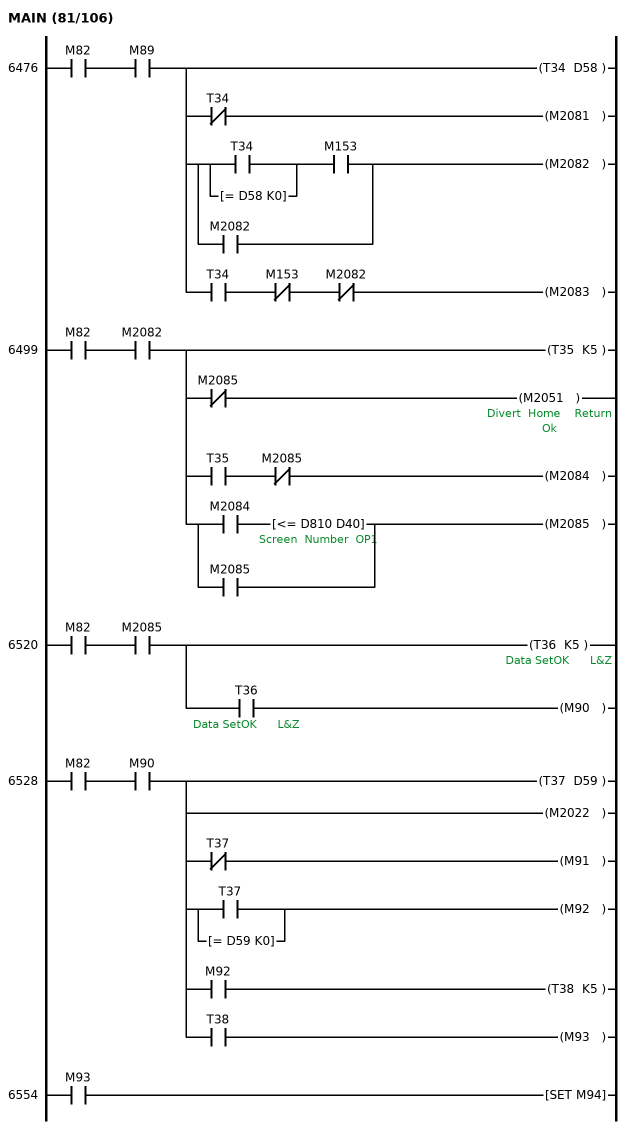
[picture p360: ladder of MAIN, rungs at steps 6476 to 6554]
6476  LD      M82
      AND     M89
      OUT     T34 D58
      MPS
      ANI     T34
      OUT     M2081
      MRD
      LD      T34
      OR=     D58 K0
      AND     M153
      OR      M2082
      ANB
      OUT     M2082
      MPP
      AND     T34
      ANI     M153
      ANI     M2082
      OUT     M2083
6499  LD      M82
      AND     M2082
      OUT     T35 K5
      MPS
      ANI     M2085
      OUT     M2051  ; Divert  Home    Return  Ok
      MRD
      AND     T35
      ANI     M2085
      OUT     M2084
      MPP
      LD      M2084
      AND<=   D810 D40  ; Screen  Number  OP1
      OR      M2085
      ANB
      OUT     M2085
6520  LD      M82
      AND     M2085
      OUT     T36 K5  ; Data SetOK      L&Z
      AND     T36  ; Data SetOK      L&Z
      OUT     M90
6528  LD      M82
      AND     M90
      OUT     T37 D59
      OUT     M2022
      MPS
      ANI     T37
      OUT     M91
      MRD
      LD      T37
      OR=     D59 K0
      ANB
      OUT     M92
      MRD
      AND     M92
      OUT     T38 K5
      MPP
      AND     T38
      OUT     M93
6554  LD      M93
      SET     M94
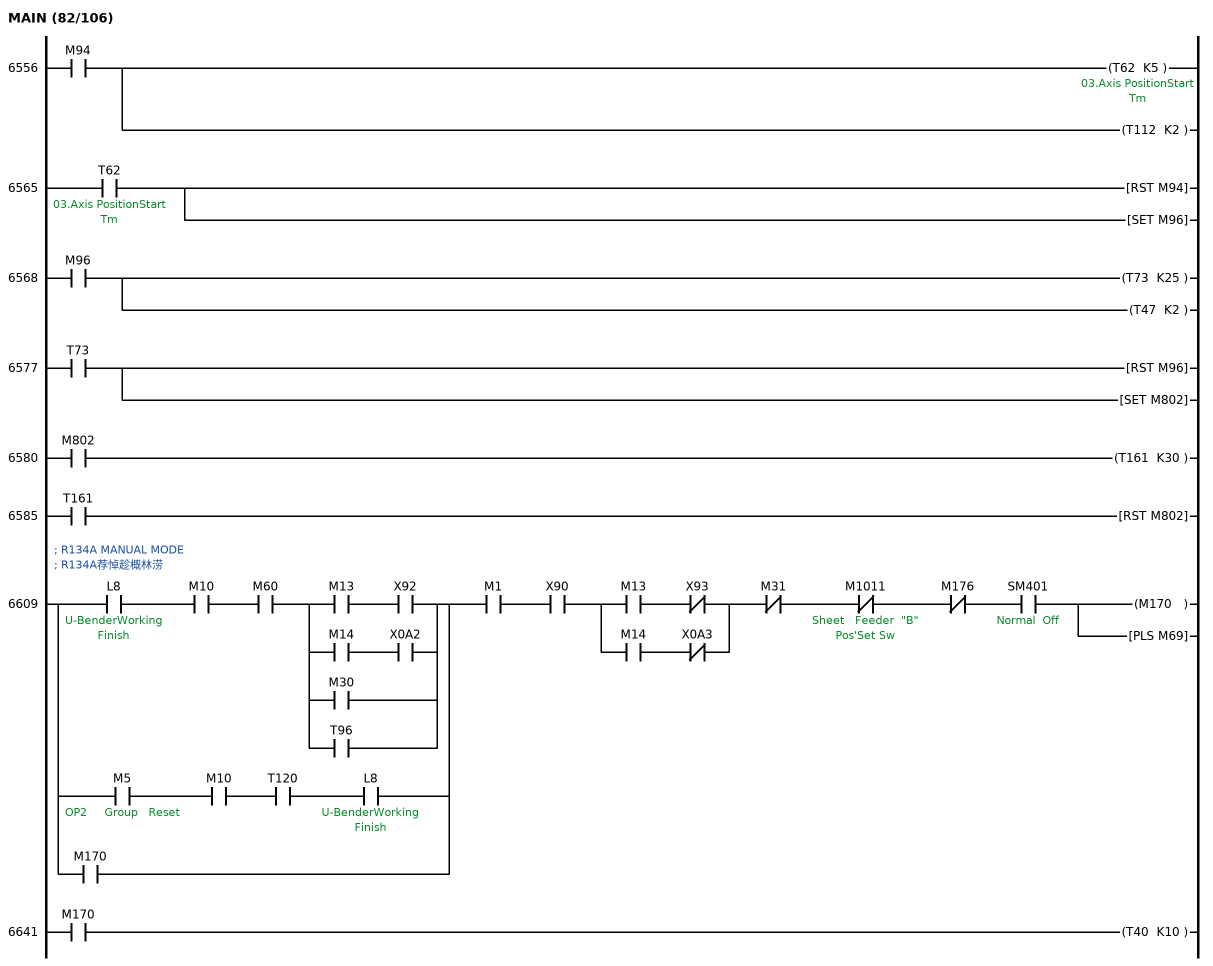
6556  LD      M94
      OUT     T62 K5  ; 03.Axis PositionStart Tm
      OUT     T112 K2
6565  LD      T62  ; 03.Axis PositionStart Tm
      RST     M94
      SET     M96
6568  LD      M96
      OUT     T73 K25
      OUT     T47 K2
6577  LD      T73
      RST     M96
      SET     M802
6580  LD      M802
      OUT     T161 K30
6585  LD      T161
      RST     M802
; R134A MANUAL MODE
; R134A수동냉매주입
6609  LD      L8  ; U-BenderWorking Finish
      AND     M10
      AND     M60
      LD      M13
      AND     X92
      LD      M14
      AND     X0A2
      ORB
      OR      M30
      OR      T96
      ANB
      LD      M5  ; OP2     Group   Reset
      AND     M10
      AND     T120
      AND     L8  ; U-BenderWorking Finish
      ORB
      OR      M170
      AND     M1
      AND     X90
      LD      M13
      ANI     X93
      LD      M14
      ANI     X0A3
      ORB
      ANB
      ANI     M31
      ANI     M1011  ; Sheet   Feeder  "B" Pos'Set Sw
      ANI     M176
      AND     SM401  ; Normal  Off
      OUT     M170
      PLS     M69
6641  LD      M170
      OUT     T40 K10
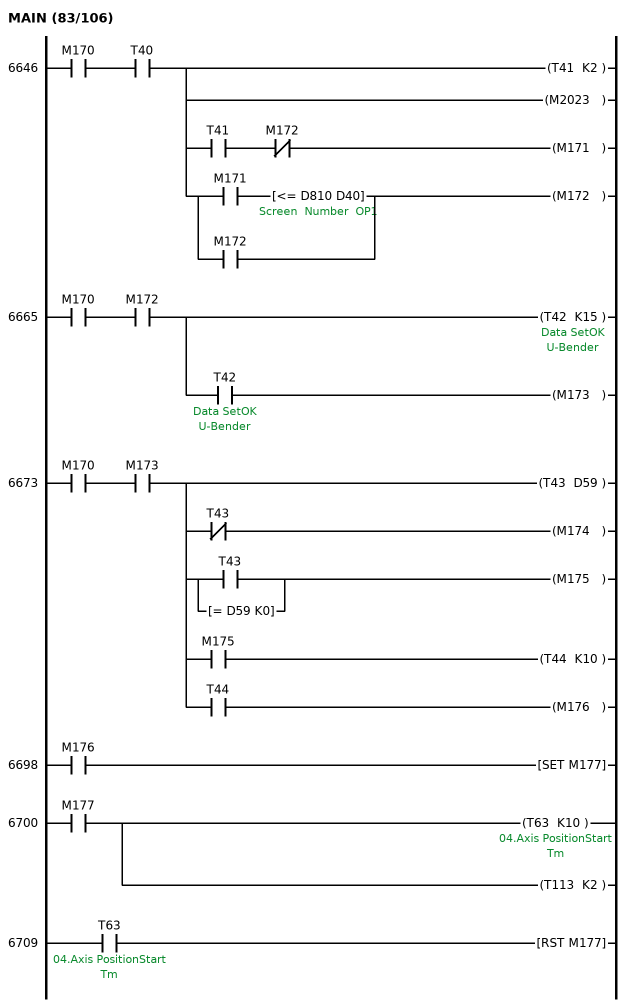
6646  LD      M170
      AND     T40
      OUT     T41 K2
      OUT     M2023
      MPS
      AND     T41
      ANI     M172
      OUT     M171
      MPP
      LD      M171
      AND<=   D810 D40  ; Screen  Number  OP1
      OR      M172
      ANB
      OUT     M172
6665  LD      M170
      AND     M172
      OUT     T42 K15  ; Data SetOK      U-Bender
      AND     T42  ; Data SetOK      U-Bender
      OUT     M173
6673  LD      M170
      AND     M173
      OUT     T43 D59
      MPS
      ANI     T43
      OUT     M174
      MRD
      LD      T43
      OR=     D59 K0
      ANB
      OUT     M175
      MRD
      AND     M175
      OUT     T44 K10
      MPP
      AND     T44
      OUT     M176
6698  LD      M176
      SET     M177
6700  LD      M177
      OUT     T63 K10  ; 04.Axis PositionStart Tm
      OUT     T113 K2
6709  LD      T63  ; 04.Axis PositionStart Tm
      RST     M177
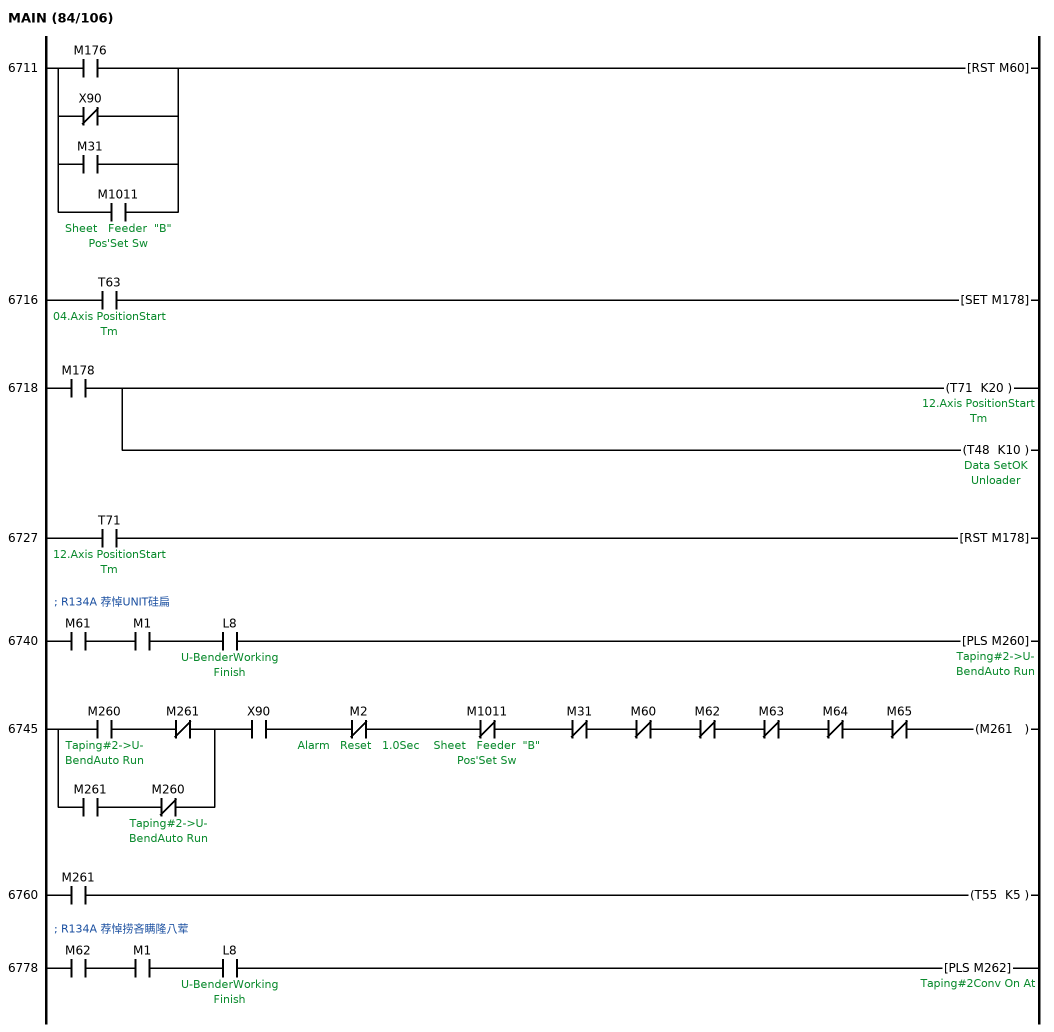
6711  LD      M176
      ORI     X90
      OR      M31
      OR      M1011  ; Sheet   Feeder  "B" Pos'Set Sw
      RST     M60
6716  LD      T63  ; 04.Axis PositionStart Tm
      SET     M178
6718  LD      M178
      OUT     T71 K20  ; 12.Axis PositionStart Tm
      OUT     T48 K10  ; Data SetOK      Unloader
6727  LD      T71  ; 12.Axis PositionStart Tm
      RST     M178
; R134A 수동UNIT배기
6740  LD      M61
      AND     M1
      AND     L8  ; U-BenderWorking Finish
      PLS     M260  ; Taping#2->U-BendAuto Run
6745  LD      M260  ; Taping#2->U-BendAuto Run
      ANI     M261
      LD      M261
      ANI     M260  ; Taping#2->U-BendAuto Run
      ORB
      AND     X90
      ANI     M2  ; Alarm   Reset   1.0Sec
      ANI     M1011  ; Sheet   Feeder  "B" Pos'Set Sw
      ANI     M31
      ANI     M60
      ANI     M62
      ANI     M63
      ANI     M64
      ANI     M65
      OUT     M261
6760  LD      M261
      OUT     T55 K5
; R134A 수동이중차징검사
6778  LD      M62
      AND     M1
      AND     L8  ; U-BenderWorking Finish
      PLS     M262  ; Taping#2Conv On At
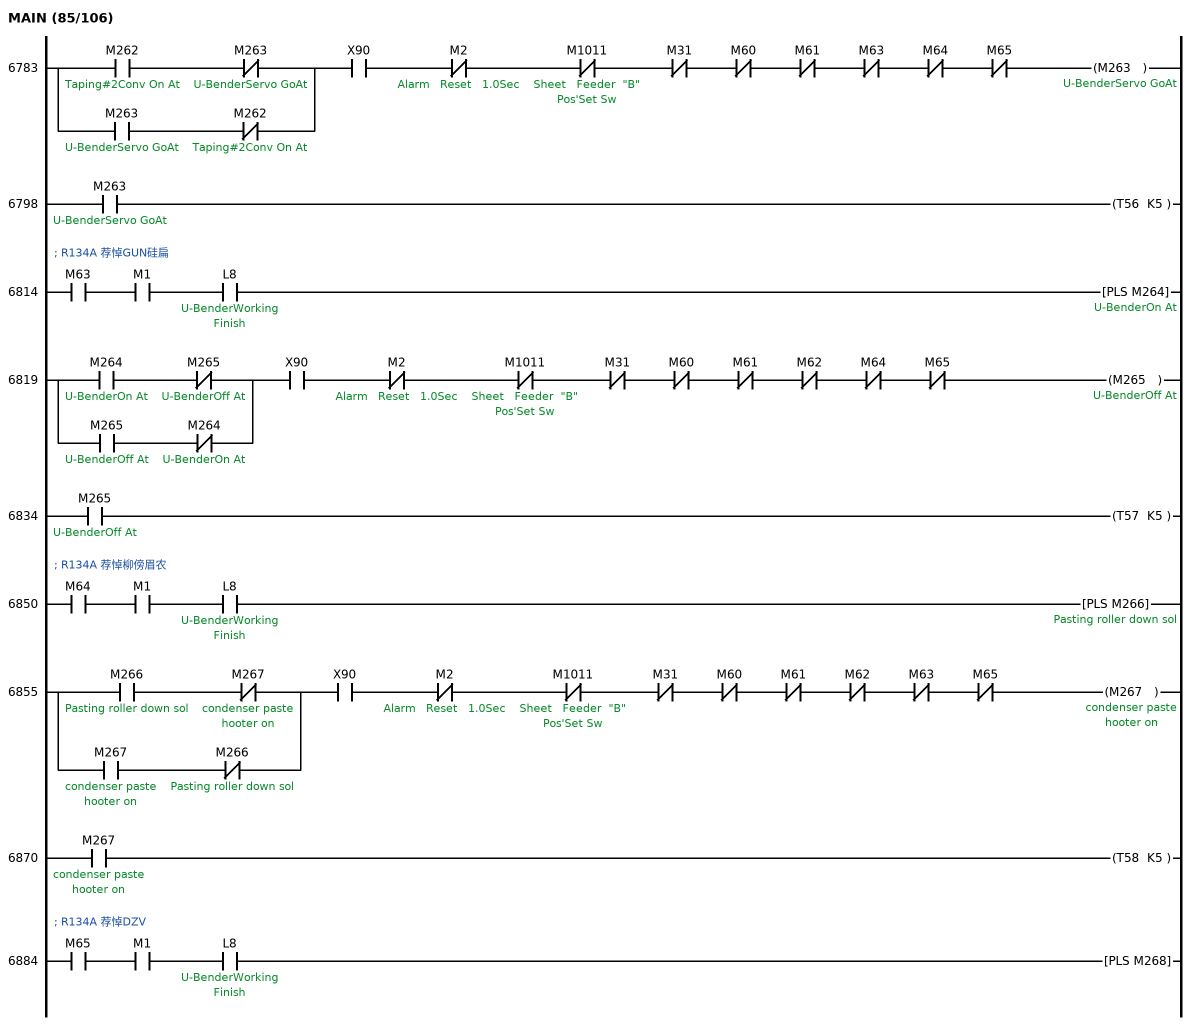
6783  LD      M262  ; Taping#2Conv On At
      ANI     M263  ; U-BenderServo GoAt
      LD      M263  ; U-BenderServo GoAt
      ANI     M262  ; Taping#2Conv On At
      ORB
      AND     X90
      ANI     M2  ; Alarm   Reset   1.0Sec
      ANI     M1011  ; Sheet   Feeder  "B" Pos'Set Sw
      ANI     M31
      ANI     M60
      ANI     M61
      ANI     M63
      ANI     M64
      ANI     M65
      OUT     M263  ; U-BenderServo GoAt
6798  LD      M263  ; U-BenderServo GoAt
      OUT     T56 K5
; R134A 수동GUN배기
6814  LD      M63
      AND     M1
      AND     L8  ; U-BenderWorking Finish
      PLS     M264  ; U-BenderOn At
6819  LD      M264  ; U-BenderOn At
      ANI     M265  ; U-BenderOff At
      LD      M265  ; U-BenderOff At
      ANI     M264  ; U-BenderOn At
      ORB
      AND     X90
      ANI     M2  ; Alarm   Reset   1.0Sec
      ANI     M1011  ; Sheet   Feeder  "B" Pos'Set Sw
      ANI     M31
      ANI     M60
      ANI     M61
      ANI     M62
      ANI     M64
      ANI     M65
      OUT     M265  ; U-BenderOff At
6834  LD      M265  ; U-BenderOff At
      OUT     T57 K5
; R134A 수동진공체크
6850  LD      M64
      AND     M1
      AND     L8  ; U-BenderWorking Finish
      PLS     M266  ; Pasting roller down sol
6855  LD      M266  ; Pasting roller down sol
      ANI     M267  ; condenser paste hooter on
      LD      M267  ; condenser paste hooter on
      ANI     M266  ; Pasting roller down sol
      ORB
      AND     X90
      ANI     M2  ; Alarm   Reset   1.0Sec
      ANI     M1011  ; Sheet   Feeder  "B" Pos'Set Sw
      ANI     M31
      ANI     M60
      ANI     M61
      ANI     M62
      ANI     M63
      ANI     M65
      OUT     M267  ; condenser paste hooter on
6870  LD      M267  ; condenser paste hooter on
      OUT     T58 K5
; R134A 수동DZV
6884  LD      M65
      AND     M1
      AND     L8  ; U-BenderWorking Finish
      PLS     M268
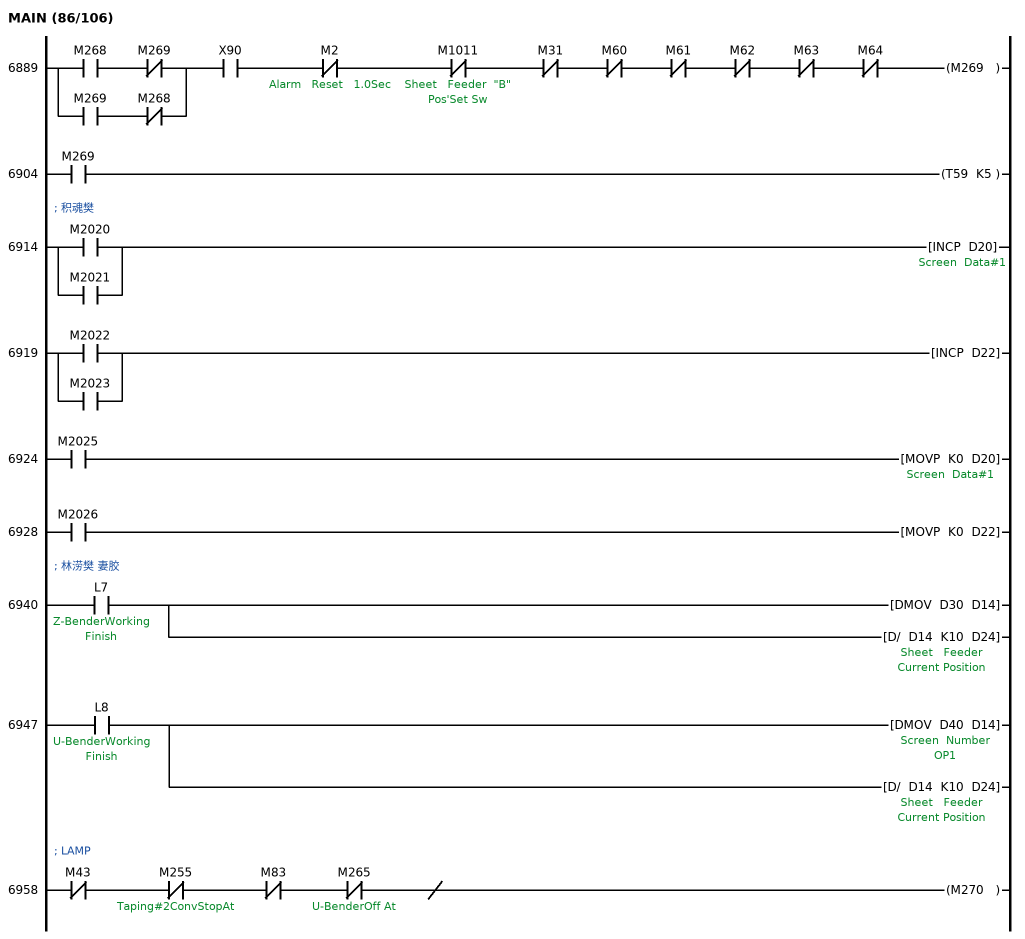
6889  LD      M268
      ANI     M269
      LD      M269
      ANI     M268
      ORB
      AND     X90
      ANI     M2  ; Alarm   Reset   1.0Sec
      ANI     M1011  ; Sheet   Feeder  "B" Pos'Set Sw
      ANI     M31
      ANI     M60
      ANI     M61
      ANI     M62
      ANI     M63
      ANI     M64
      OUT     M269
6904  LD      M269
      OUT     T59 K5
; 积魂樊
6914  LD      M2020
      OR      M2021
      INCP    D20  ; Screen  Data#1
6919  LD      M2022
      OR      M2023
      INCP    D22
6924  LD      M2025
      MOVP    K0 D20
6928  LD      M2026
      MOVP    K0 D22
; 주입량 펄스
6940  LD      L7  ; Z-BenderWorking Finish
      DMOV    D30 D14
      D/      D14 K10 D24  ; Sheet   Feeder  Current Position
6947  LD      L8  ; U-BenderWorking Finish
      DMOV    D40 D14
      D/      D14 K10 D24
; LAMP
6958  LDI     M43
      ANI     M255  ; Taping#2ConvStopAt
      ANI     M83
      ANI     M265  ; U-BenderOff At
      INV
      OUT     M270
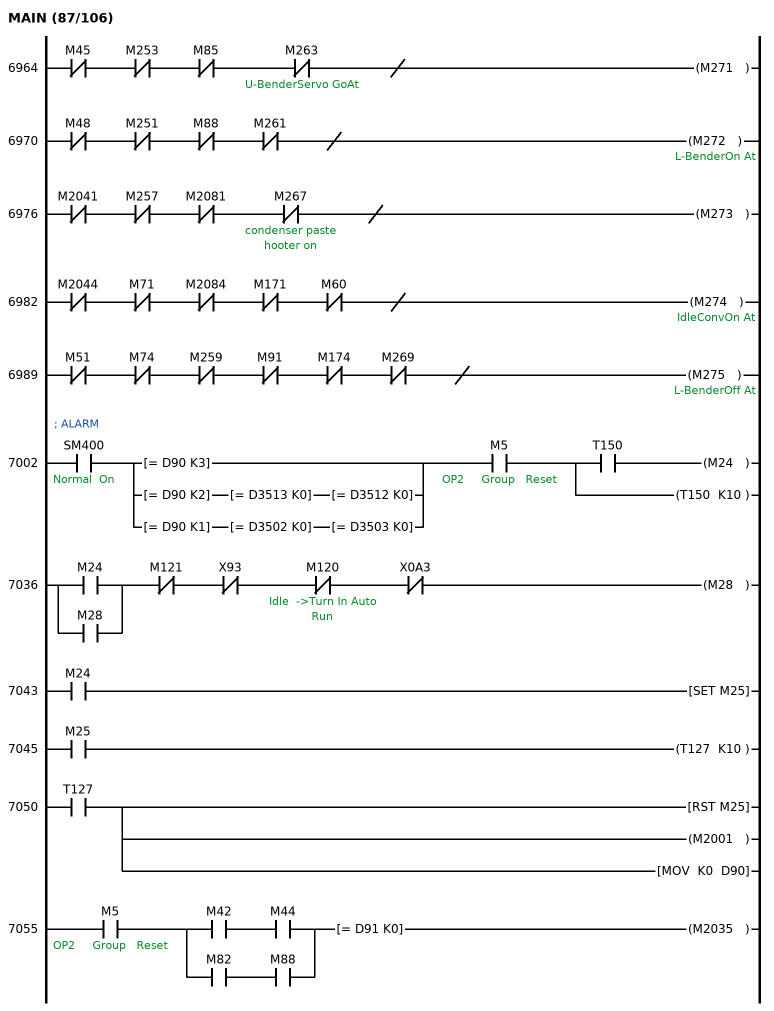
6964  LDI     M45
      ANI     M253
      ANI     M85
      ANI     M263  ; U-BenderServo GoAt
      INV
      OUT     M271
6970  LDI     M48
      ANI     M251
      ANI     M88
      ANI     M261
      INV
      OUT     M272  ; L-BenderOn At
6976  LDI     M2041
      ANI     M257
      ANI     M2081
      ANI     M267  ; condenser paste hooter on
      INV
      OUT     M273
6982  LDI     M2044
      ANI     M71
      ANI     M2084
      ANI     M171
      ANI     M60
      INV
      OUT     M274  ; IdleConvOn At
6989  LDI     M51
      ANI     M74
      ANI     M259
      ANI     M91
      ANI     M174
      ANI     M269
      INV
      OUT     M275  ; L-BenderOff At
; ALARM
7002  LD      SM400  ; Normal  On
      LD=     D90 K3
      LD=     D90 K2
      AND=    D3513 K0
      AND=    D3512 K0
      ORB
      LD=     D90 K1
      AND=    D3502 K0
      AND=    D3503 K0
      ORB
      ANB
      AND     M5  ; OP2     Group   Reset
      MPS
      AND     T150
      OUT     M24
      MPP
      OUT     T150 K10
7036  LD      M24
      OR      M28
      ANI     M121
      ANI     X93
      ANI     M120  ; Idle  ->Turn In Auto Run
      ANI     X0A3
      OUT     M28
7043  LD      M24
      SET     M25
7045  LD      M25
      OUT     T127 K10
7050  LD      T127
      RST     M25
      OUT     M2001
      MOV     K0 D90
7055  LD      M5  ; OP2     Group   Reset
      LD      M42
      AND     M44
      LD      M82
      AND     M88
      ORB
      ANB
      AND=    D91 K0
      OUT     M2035
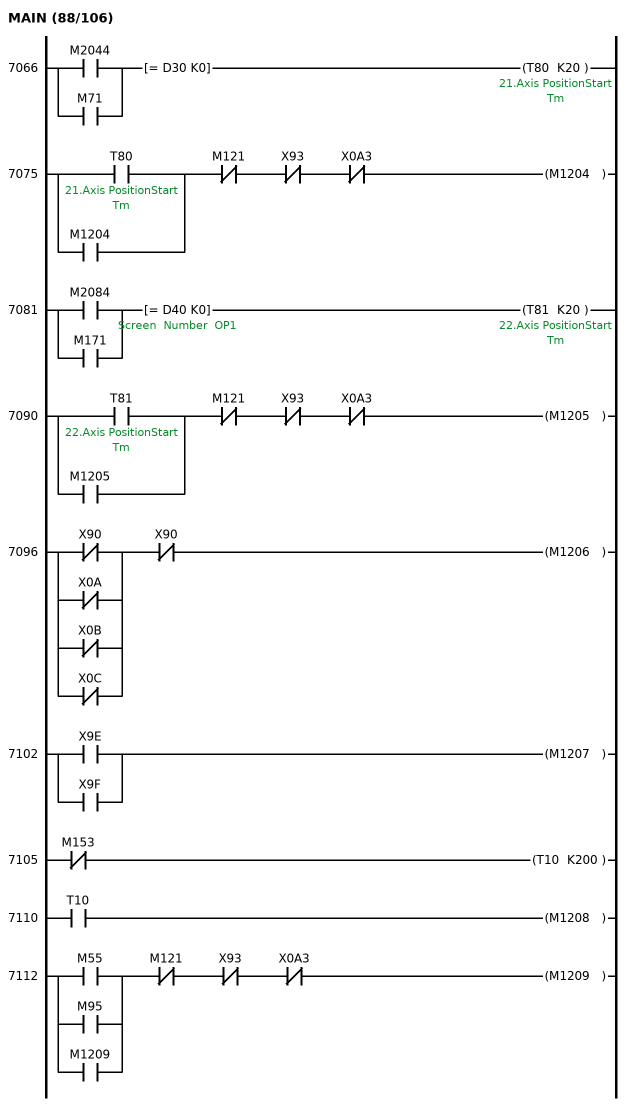
7066  LD      M2044
      OR      M71
      AND=    D30 K0
      OUT     T80 K20  ; 21.Axis PositionStart Tm
7075  LD      T80  ; 21.Axis PositionStart Tm
      OR      M1204
      ANI     M121
      ANI     X93
      ANI     X0A3
      OUT     M1204
7081  LD      M2084
      OR      M171
      AND=    D40 K0  ; Screen  Number  OP1
      OUT     T81 K20  ; 22.Axis PositionStart Tm
7090  LD      T81  ; 22.Axis PositionStart Tm
      OR      M1205
      ANI     M121
      ANI     X93
      ANI     X0A3
      OUT     M1205
7096  LDI     X90
      ORI     X0A
      ORI     X0B
      ORI     X0C
      ANI     X90
      OUT     M1206
7102  LD      X9E
      OR      X9F
      OUT     M1207
7105  LDI     M153
      OUT     T10 K200
7110  LD      T10
      OUT     M1208
7112  LD      M55
      OR      M95
      OR      M1209
      ANI     M121
      ANI     X93
      ANI     X0A3
      OUT     M1209
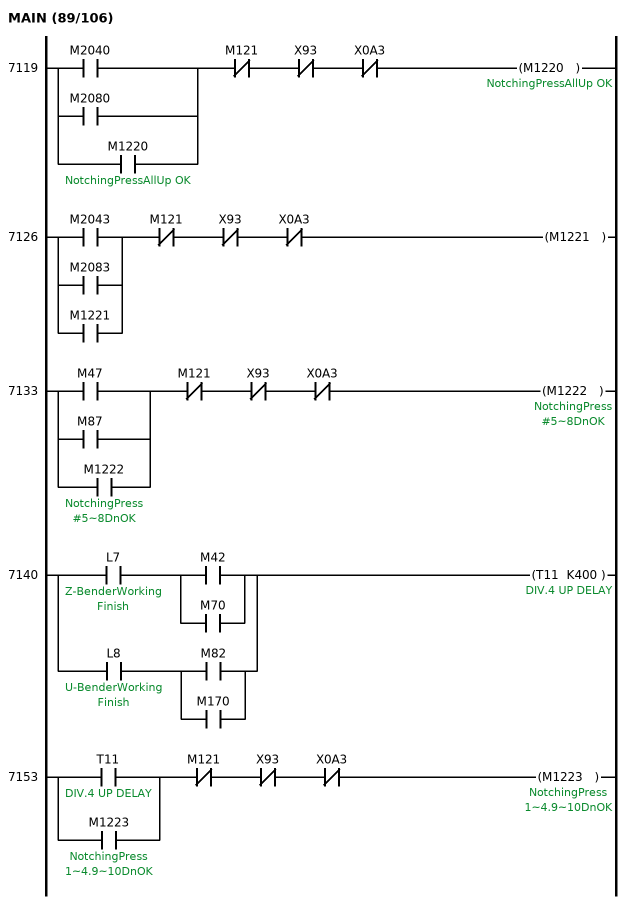
7119  LD      M2040
      OR      M2080
      OR      M1220  ; NotchingPressAllUp OK
      ANI     M121
      ANI     X93
      ANI     X0A3
      OUT     M1220  ; NotchingPressAllUp OK
7126  LD      M2043
      OR      M2083
      OR      M1221
      ANI     M121
      ANI     X93
      ANI     X0A3
      OUT     M1221
7133  LD      M47
      OR      M87
      OR      M1222  ; NotchingPress   #5~8DnOK
      ANI     M121
      ANI     X93
      ANI     X0A3
      OUT     M1222  ; NotchingPress   #5~8DnOK
7140  LD      L7  ; Z-BenderWorking Finish
      LD      M42
      OR      M70
      ANB
      LD      L8  ; U-BenderWorking Finish
      LD      M82
      OR      M170
      ANB
      ORB
      OUT     T11 K400  ; DIV.4 UP DELAY
7153  LD      T11  ; DIV.4 UP DELAY
      OR      M1223  ; NotchingPress   1~4.9~10DnOK
      ANI     M121
      ANI     X93
      ANI     X0A3
      OUT     M1223  ; NotchingPress   1~4.9~10DnOK
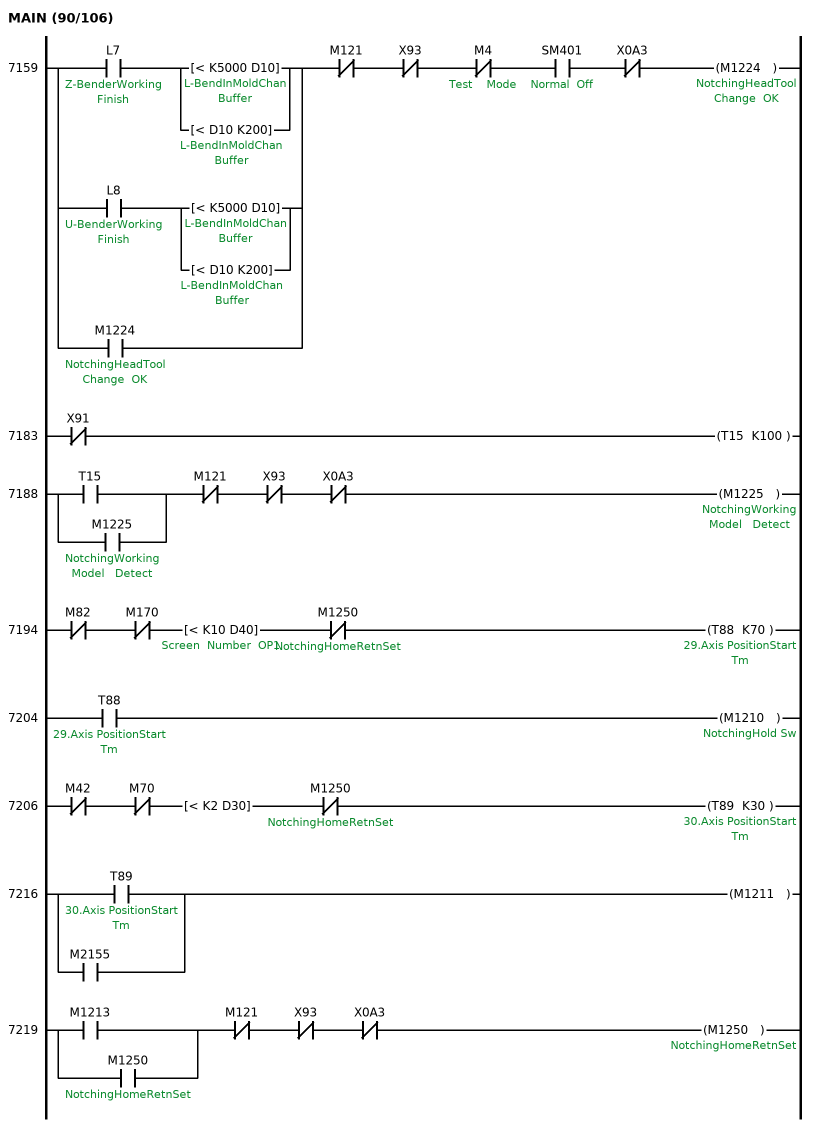
7159  LD      L7  ; Z-BenderWorking Finish
      LD<     K5000 D10  ; L-BendInMoldChanBuffer
      OR<     D10 K200  ; L-BendInMoldChanBuffer
      ANB
      LD      L8  ; U-BenderWorking Finish
      LD<     K5000 D10  ; L-BendInMoldChanBuffer
      OR<     D10 K200  ; L-BendInMoldChanBuffer
      ANB
      ORB
      OR      M1224  ; NotchingHeadToolChange  OK
      ANI     M121
      ANI     X93
      ANI     M4  ; Test    Mode
      AND     SM401  ; Normal  Off
      ANI     X0A3
      OUT     M1224  ; NotchingHeadToolChange  OK
7183  LDI     X91
      OUT     T15 K100
7188  LD      T15
      OR      M1225  ; NotchingWorking Model   Detect
      ANI     M121
      ANI     X93
      ANI     X0A3
      OUT     M1225  ; NotchingWorking Model   Detect
7194  LDI     M82
      ANI     M170
      AND<    K10 D40  ; Screen  Number  OP1
      ANI     M1250  ; NotchingHomeRetnSet
      OUT     T88 K70  ; 29.Axis PositionStart Tm
7204  LD      T88  ; 29.Axis PositionStart Tm
      OUT     M1210  ; NotchingHold Sw
7206  LDI     M42
      ANI     M70
      AND<    K2 D30
      ANI     M1250  ; NotchingHomeRetnSet
      OUT     T89 K30  ; 30.Axis PositionStart Tm
7216  LD      T89  ; 30.Axis PositionStart Tm
      OR      M2155
      OUT     M1211
7219  LD      M1213
      OR      M1250  ; NotchingHomeRetnSet
      ANI     M121
      ANI     X93
      ANI     X0A3
      OUT     M1250  ; NotchingHomeRetnSet
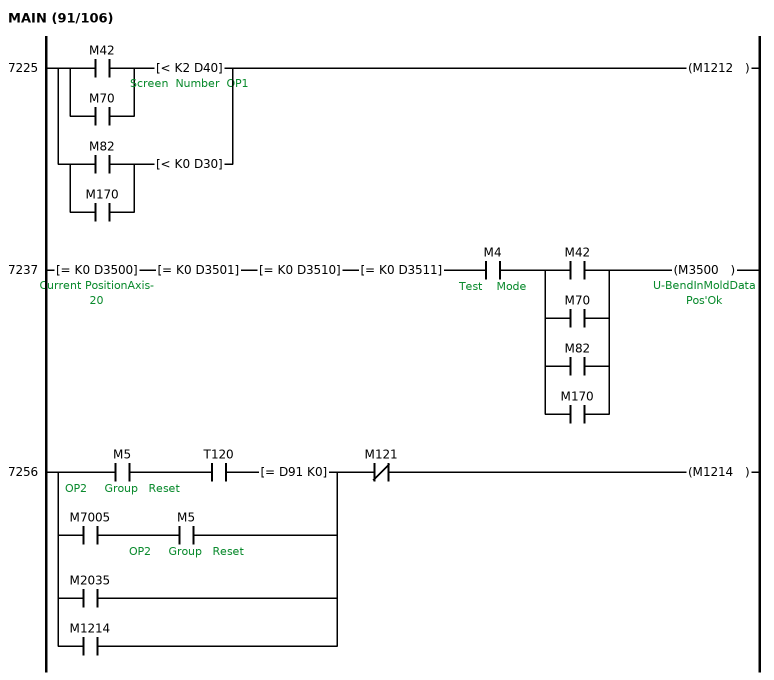
7225  LD      M42
      OR      M70
      AND<    K2 D40  ; Screen  Number  OP1
      LD      M82
      OR      M170
      AND<    K0 D30
      ORB
      OUT     M1212
7237  LD=     K0 D3500  ; Current PositionAxis-20
      AND=    K0 D3501
      AND=    K0 D3510
      AND=    K0 D3511
      AND     M4  ; Test    Mode
      LD      M42
      OR      M70
      OR      M82
      OR      M170
      ANB
      OUT     M3500  ; U-BendInMoldDataPos'Ok
7256  LD      M5  ; OP2     Group   Reset
      AND     T120
      AND=    D91 K0
      LD      M7005
      AND     M5  ; OP2     Group   Reset
      ORB
      OR      M2035
      OR      M1214
      ANI     M121
      OUT     M1214
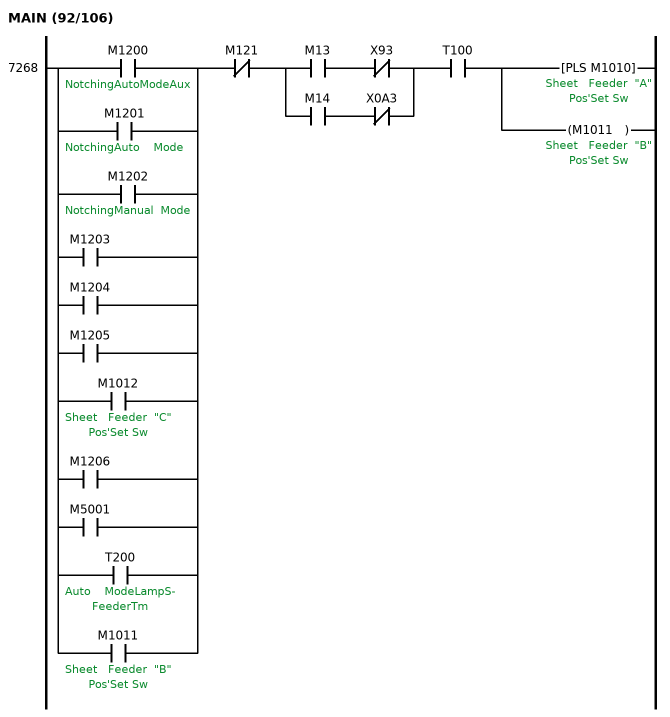
7268  LD      M1200  ; NotchingAutoModeAux
      OR      M1201  ; NotchingAuto    Mode
      OR      M1202  ; NotchingManual  Mode
      OR      M1203
      OR      M1204
      OR      M1205
      OR      M1012  ; Sheet   Feeder  "C" Pos'Set Sw
      OR      M1206
      OR      M5001
      OR      T200  ; Auto    ModeLampS-FeederTm
      OR      M1011  ; Sheet   Feeder  "B" Pos'Set Sw
      ANI     M121
      LD      M13
      ANI     X93
      LD      M14
      ANI     X0A3
      ORB
      ANB
      AND     T100
      PLS     M1010  ; Sheet   Feeder  "A" Pos'Set Sw
      OUT     M1011  ; Sheet   Feeder  "B" Pos'Set Sw
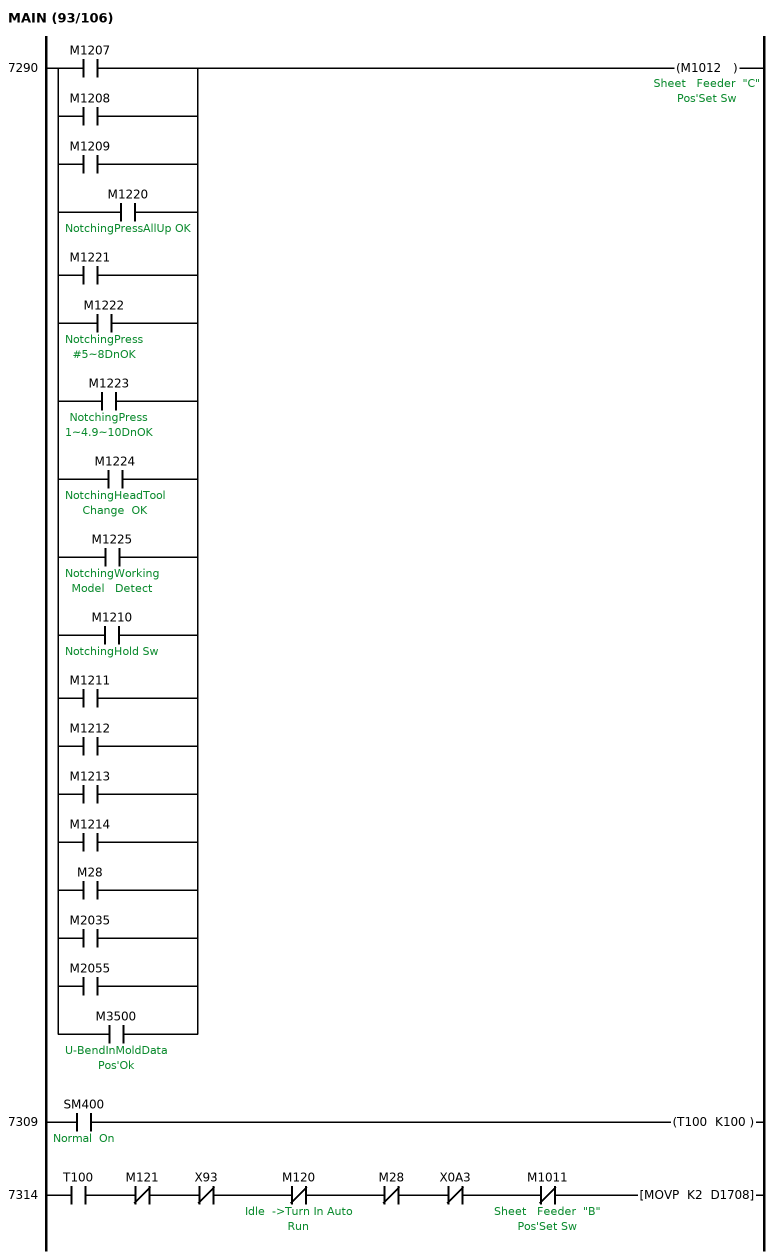
7290  LD      M1207
      OR      M1208
      OR      M1209
      OR      M1220  ; NotchingPressAllUp OK
      OR      M1221
      OR      M1222  ; NotchingPress   #5~8DnOK
      OR      M1223  ; NotchingPress   1~4.9~10DnOK
      OR      M1224  ; NotchingHeadToolChange  OK
      OR      M1225  ; NotchingWorking Model   Detect
      OR      M1210  ; NotchingHold Sw
      OR      M1211
      OR      M1212
      OR      M1213
      OR      M1214
      OR      M28
      OR      M2035
      OR      M2055
      OR      M3500  ; U-BendInMoldDataPos'Ok
      OUT     M1012  ; Sheet   Feeder  "C" Pos'Set Sw
7309  LD      SM400  ; Normal  On
      OUT     T100 K100
7314  LD      T100
      ANI     M121
      ANI     X93
      ANI     M120  ; Idle  ->Turn In Auto Run
      ANI     M28
      ANI     X0A3
      ANI     M1011  ; Sheet   Feeder  "B" Pos'Set Sw
      MOVP    K2 D1708
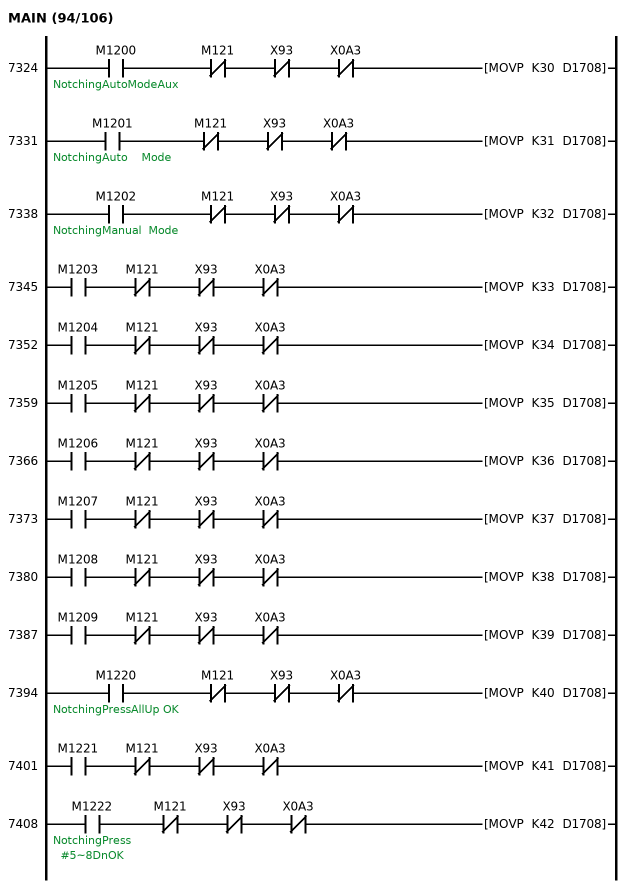
7324  LD      M1200  ; NotchingAutoModeAux
      ANI     M121
      ANI     X93
      ANI     X0A3
      MOVP    K30 D1708
7331  LD      M1201  ; NotchingAuto    Mode
      ANI     M121
      ANI     X93
      ANI     X0A3
      MOVP    K31 D1708
7338  LD      M1202  ; NotchingManual  Mode
      ANI     M121
      ANI     X93
      ANI     X0A3
      MOVP    K32 D1708
7345  LD      M1203
      ANI     M121
      ANI     X93
      ANI     X0A3
      MOVP    K33 D1708
7352  LD      M1204
      ANI     M121
      ANI     X93
      ANI     X0A3
      MOVP    K34 D1708
7359  LD      M1205
      ANI     M121
      ANI     X93
      ANI     X0A3
      MOVP    K35 D1708
7366  LD      M1206
      ANI     M121
      ANI     X93
      ANI     X0A3
      MOVP    K36 D1708
7373  LD      M1207
      ANI     M121
      ANI     X93
      ANI     X0A3
      MOVP    K37 D1708
7380  LD      M1208
      ANI     M121
      ANI     X93
      ANI     X0A3
      MOVP    K38 D1708
7387  LD      M1209
      ANI     M121
      ANI     X93
      ANI     X0A3
      MOVP    K39 D1708
7394  LD      M1220  ; NotchingPressAllUp OK
      ANI     M121
      ANI     X93
      ANI     X0A3
      MOVP    K40 D1708
7401  LD      M1221
      ANI     M121
      ANI     X93
      ANI     X0A3
      MOVP    K41 D1708
7408  LD      M1222  ; NotchingPress   #5~8DnOK
      ANI     M121
      ANI     X93
      ANI     X0A3
      MOVP    K42 D1708
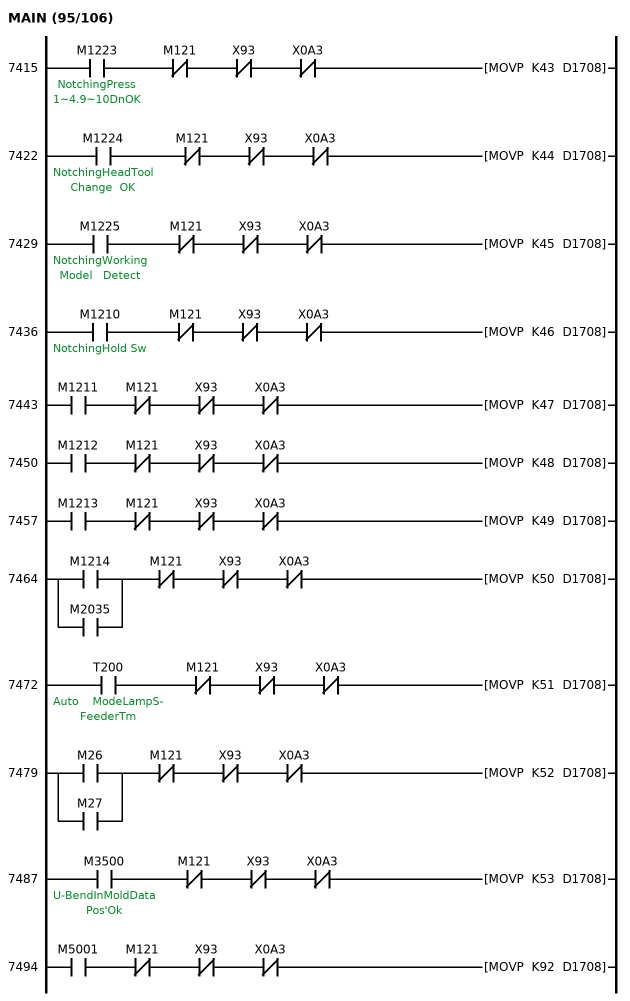
7415  LD      M1223  ; NotchingPress   1~4.9~10DnOK
      ANI     M121
      ANI     X93
      ANI     X0A3
      MOVP    K43 D1708
7422  LD      M1224  ; NotchingHeadToolChange  OK
      ANI     M121
      ANI     X93
      ANI     X0A3
      MOVP    K44 D1708
7429  LD      M1225  ; NotchingWorking Model   Detect
      ANI     M121
      ANI     X93
      ANI     X0A3
      MOVP    K45 D1708
7436  LD      M1210  ; NotchingHold Sw
      ANI     M121
      ANI     X93
      ANI     X0A3
      MOVP    K46 D1708
7443  LD      M1211
      ANI     M121
      ANI     X93
      ANI     X0A3
      MOVP    K47 D1708
7450  LD      M1212
      ANI     M121
      ANI     X93
      ANI     X0A3
      MOVP    K48 D1708
7457  LD      M1213
      ANI     M121
      ANI     X93
      ANI     X0A3
      MOVP    K49 D1708
7464  LD      M1214
      OR      M2035
      ANI     M121
      ANI     X93
      ANI     X0A3
      MOVP    K50 D1708
7472  LD      T200  ; Auto    ModeLampS-FeederTm
      ANI     M121
      ANI     X93
      ANI     X0A3
      MOVP    K51 D1708
7479  LD      M26
      OR      M27
      ANI     M121
      ANI     X93
      ANI     X0A3
      MOVP    K52 D1708
7487  LD      M3500  ; U-BendInMoldDataPos'Ok
      ANI     M121
      ANI     X93
      ANI     X0A3
      MOVP    K53 D1708
7494  LD      M5001
      ANI     M121
      ANI     X93
      ANI     X0A3
      MOVP    K92 D1708
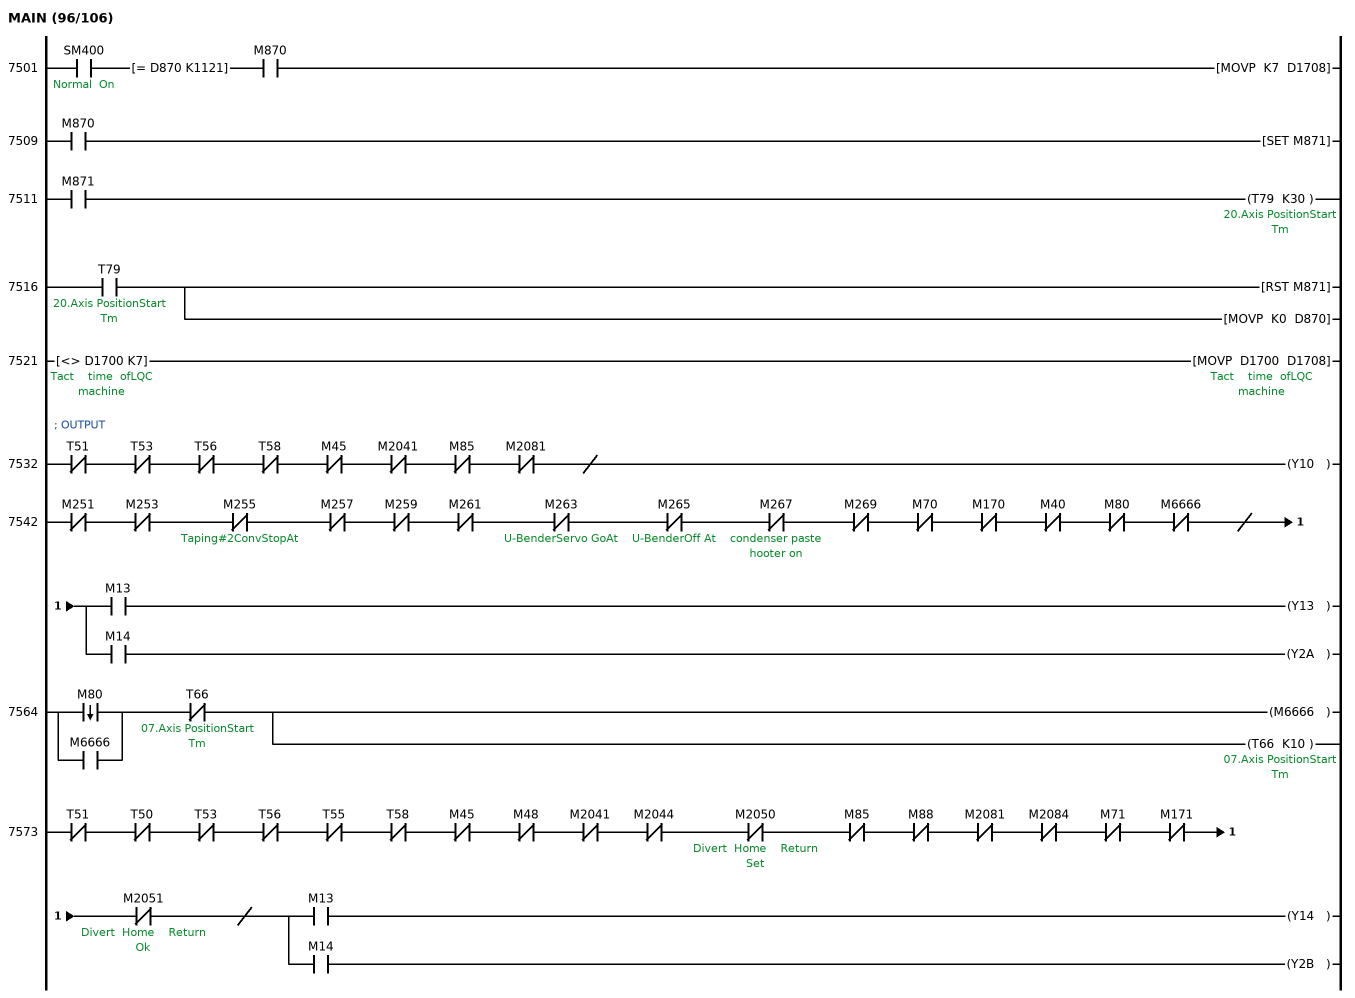
7501  LD      SM400  ; Normal  On
      AND=    D870 K1121
      AND     M870
      MOVP    K7 D1708
7509  LD      M870
      SET     M871
7511  LD      M871
      OUT     T79 K30  ; 20.Axis PositionStart Tm
7516  LD      T79  ; 20.Axis PositionStart Tm
      RST     M871
      MOVP    K0 D870
7521  LD<>    D1700 K7  ; Tact    time  ofLQC     machine
      MOVP    D1700 D1708
; OUTPUT
7532  LDI     T51
      ANI     T53
      ANI     T56
      ANI     T58
      ANI     M45
      ANI     M2041
      ANI     M85
      ANI     M2081
      INV
      OUT     Y10
7542  LDI     M251
      ANI     M253
      ANI     M255  ; Taping#2ConvStopAt
      ANI     M257
      ANI     M259
      ANI     M261
      ANI     M263  ; U-BenderServo GoAt
      ANI     M265  ; U-BenderOff At
      ANI     M267  ; condenser paste hooter on
      ANI     M269
      ANI     M70
      ANI     M170
      ANI     M40
      ANI     M80
      ANI     M6666
      INV
      MPS
      AND     M13
      OUT     Y13
      MPP
      AND     M14
      OUT     Y2A
7564  LDF     M80
      OR      M6666
      ANI     T66  ; 07.Axis PositionStart Tm
      OUT     M6666
      OUT     T66 K10  ; 07.Axis PositionStart Tm
7573  LDI     T51
      ANI     T50
      ANI     T53
      ANI     T56
      ANI     T55
      ANI     T58
      ANI     M45
      ANI     M48
      ANI     M2041
      ANI     M2044
      ANI     M2050  ; Divert  Home    Return  Set
      ANI     M85
      ANI     M88
      ANI     M2081
      ANI     M2084
      ANI     M71
      ANI     M171
      ANI     M2051  ; Divert  Home    Return  Ok
      INV
      MPS
      AND     M13
      OUT     Y14
      MPP
      AND     M14
      OUT     Y2B
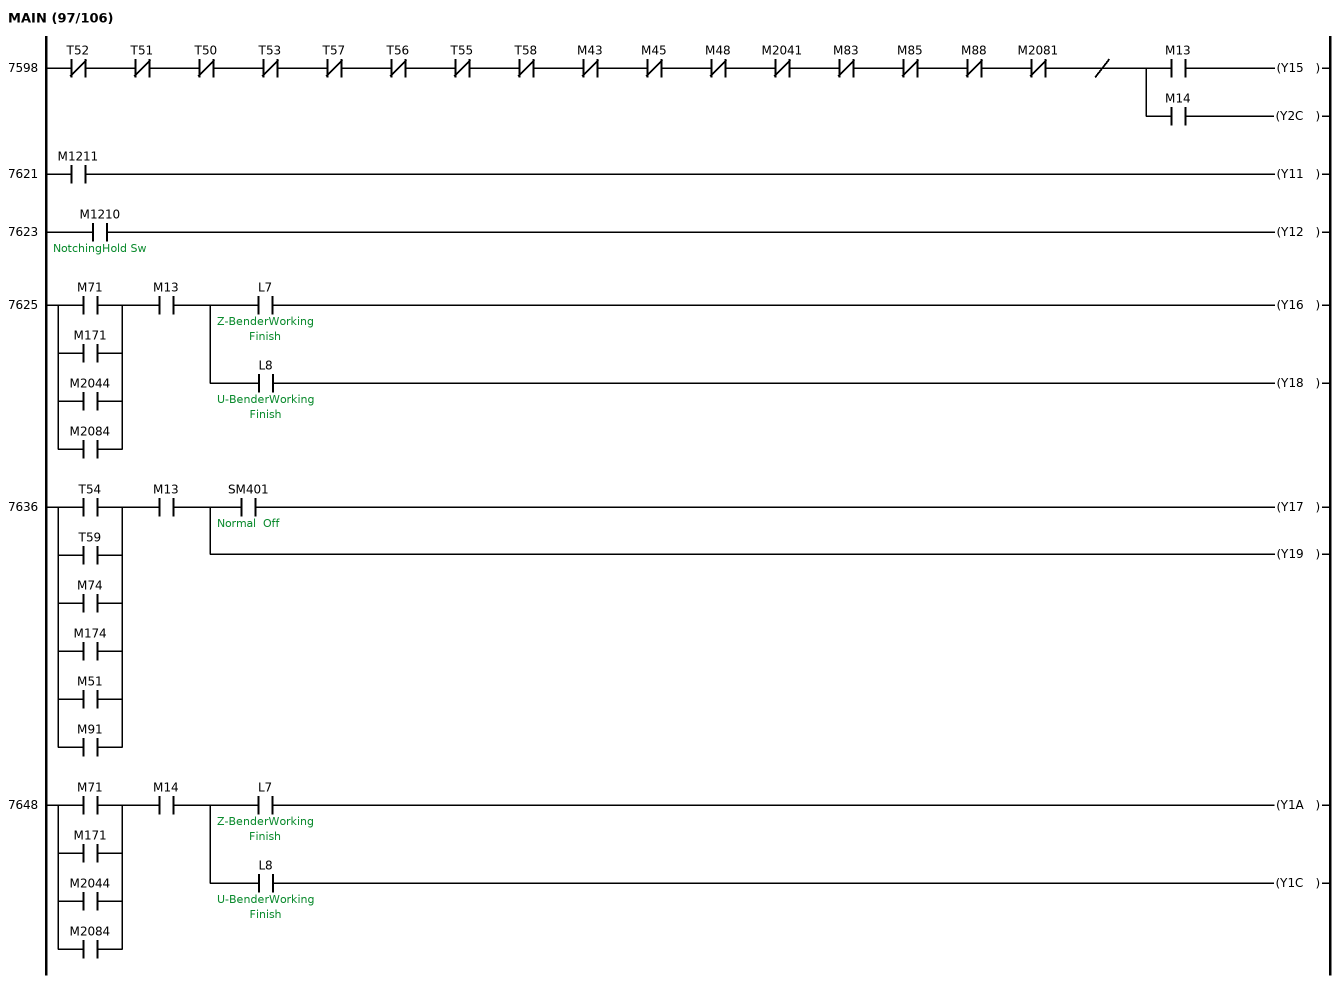
7598  LDI     T52
      ANI     T51
      ANI     T50
      ANI     T53
      ANI     T57
      ANI     T56
      ANI     T55
      ANI     T58
      ANI     M43
      ANI     M45
      ANI     M48
      ANI     M2041
      ANI     M83
      ANI     M85
      ANI     M88
      ANI     M2081
      INV
      MPS
      AND     M13
      OUT     Y15
      MPP
      AND     M14
      OUT     Y2C
7621  LD      M1211
      OUT     Y11
7623  LD      M1210  ; NotchingHold Sw
      OUT     Y12
7625  LD      M71
      OR      M171
      OR      M2044
      OR      M2084
      AND     M13
      MPS
      AND     L7  ; Z-BenderWorking Finish
      OUT     Y16
      MPP
      AND     L8  ; U-BenderWorking Finish
      OUT     Y18
7636  LD      T54
      OR      T59
      OR      M74
      OR      M174
      OR      M51
      OR      M91
      AND     M13
      MPS
      AND     SM401  ; Normal  Off
      OUT     Y17
      MPP
      OUT     Y19
7648  LD      M71
      OR      M171
      OR      M2044
      OR      M2084
      AND     M14
      MPS
      AND     L7  ; Z-BenderWorking Finish
      OUT     Y1A
      MPP
      AND     L8  ; U-BenderWorking Finish
      OUT     Y1C
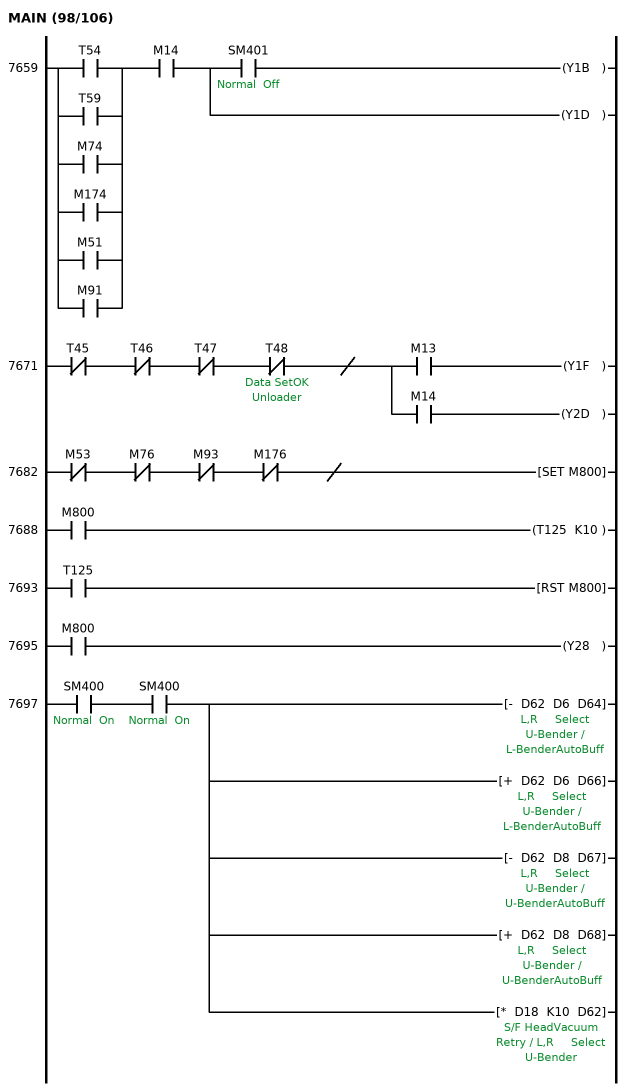
7659  LD      T54
      OR      T59
      OR      M74
      OR      M174
      OR      M51
      OR      M91
      AND     M14
      MPS
      AND     SM401  ; Normal  Off
      OUT     Y1B
      MPP
      OUT     Y1D
7671  LDI     T45
      ANI     T46
      ANI     T47
      ANI     T48  ; Data SetOK      Unloader
      INV
      MPS
      AND     M13
      OUT     Y1F
      MPP
      AND     M14
      OUT     Y2D
7682  LDI     M53
      ANI     M76
      ANI     M93
      ANI     M176
      INV
      SET     M800
7688  LD      M800
      OUT     T125 K10
7693  LD      T125
      RST     M800
7695  LD      M800
      OUT     Y28
7697  LD      SM400  ; Normal  On
      AND     SM400  ; Normal  On
      -       D62 D6 D64  ; L,R     Select  U-Bender / L-BenderAutoBuff
      +       D62 D6 D66
      -       D62 D8 D67  ; U-BenderAutoBuff
      +       D62 D8 D68
      *       D18 K10 D62
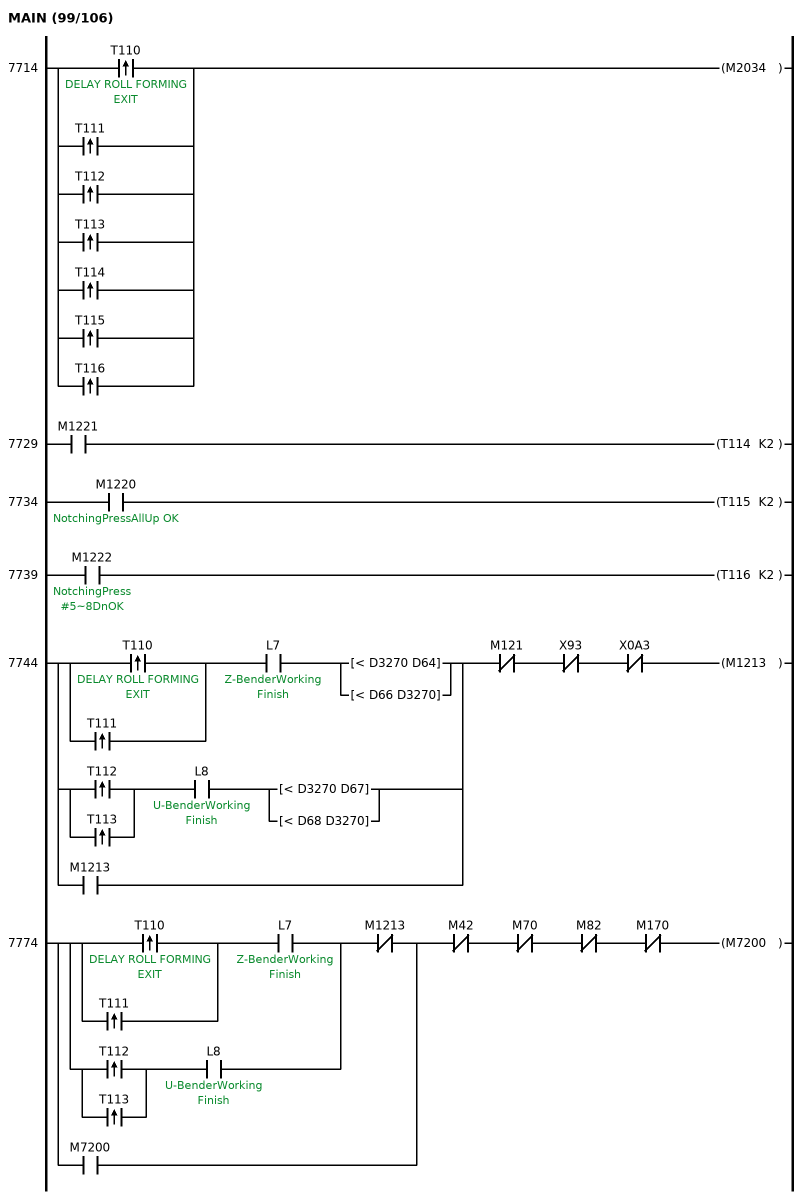
7714  LDP     T110  ; DELAY ROLL FORMING EXIT
      ORP     T111
      ORP     T112
      ORP     T113
      ORP     T114
      ORP     T115
      ORP     T116
      OUT     M2034
7729  LD      M1221
      OUT     T114 K2
7734  LD      M1220  ; NotchingPressAllUp OK
      OUT     T115 K2
7739  LD      M1222  ; NotchingPress   #5~8DnOK
      OUT     T116 K2
7744  LDP     T110  ; DELAY ROLL FORMING EXIT
      ORP     T111
      AND     L7  ; Z-BenderWorking Finish
      LD<     D3270 D64
      OR<     D66 D3270
      ANB
      LDP     T112
      ORP     T113
      AND     L8  ; U-BenderWorking Finish
      LD<     D3270 D67
      OR<     D68 D3270
      ANB
      ORB
      OR      M1213
      ANI     M121
      ANI     X93
      ANI     X0A3
      OUT     M1213
7774  LDP     T110  ; DELAY ROLL FORMING EXIT
      ORP     T111
      AND     L7  ; Z-BenderWorking Finish
      LDP     T112
      ORP     T113
      AND     L8  ; U-BenderWorking Finish
      ORB
      ANI     M1213
      OR      M7200
      ANI     M42
      ANI     M70
      ANI     M82
      ANI     M170
      OUT     M7200
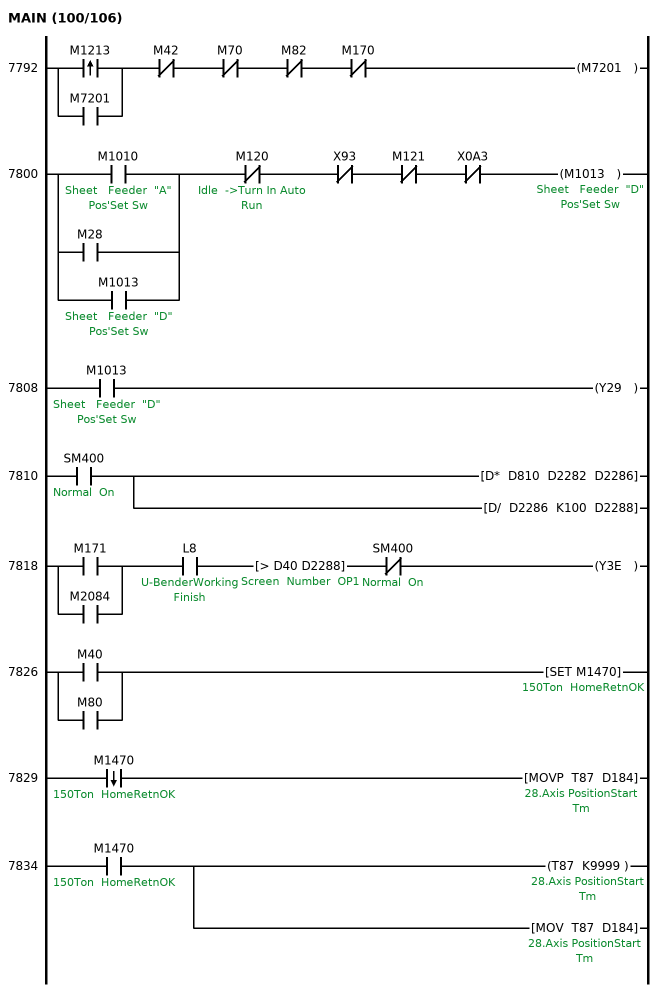
7792  LDP     M1213
      OR      M7201
      ANI     M42
      ANI     M70
      ANI     M82
      ANI     M170
      OUT     M7201
7800  LD      M1010  ; Sheet   Feeder  "A" Pos'Set Sw
      OR      M28
      OR      M1013  ; Sheet   Feeder  "D" Pos'Set Sw
      ANI     M120  ; Idle  ->Turn In Auto Run
      ANI     X93
      ANI     M121
      ANI     X0A3
      OUT     M1013  ; Sheet   Feeder  "D" Pos'Set Sw
7808  LD      M1013  ; Sheet   Feeder  "D" Pos'Set Sw
      OUT     Y29
7810  LD      SM400  ; Normal  On
      D*      D810 D2282 D2286
      D/      D2286 K100 D2288
7818  LD      M171
      OR      M2084
      AND     L8  ; U-BenderWorking Finish
      AND>    D40 D2288  ; Screen  Number  OP1
      ANI     SM400  ; Normal  On
      OUT     Y3E
7826  LD      M40
      OR      M80
      SET     M1470  ; 150Ton  HomeRetnOK
7829  LDF     M1470  ; 150Ton  HomeRetnOK
      MOVP    T87 D184  ; 28.Axis PositionStart Tm
7834  LD      M1470  ; 150Ton  HomeRetnOK
      OUT     T87 K9999  ; 28.Axis PositionStart Tm
      MOV     T87 D184
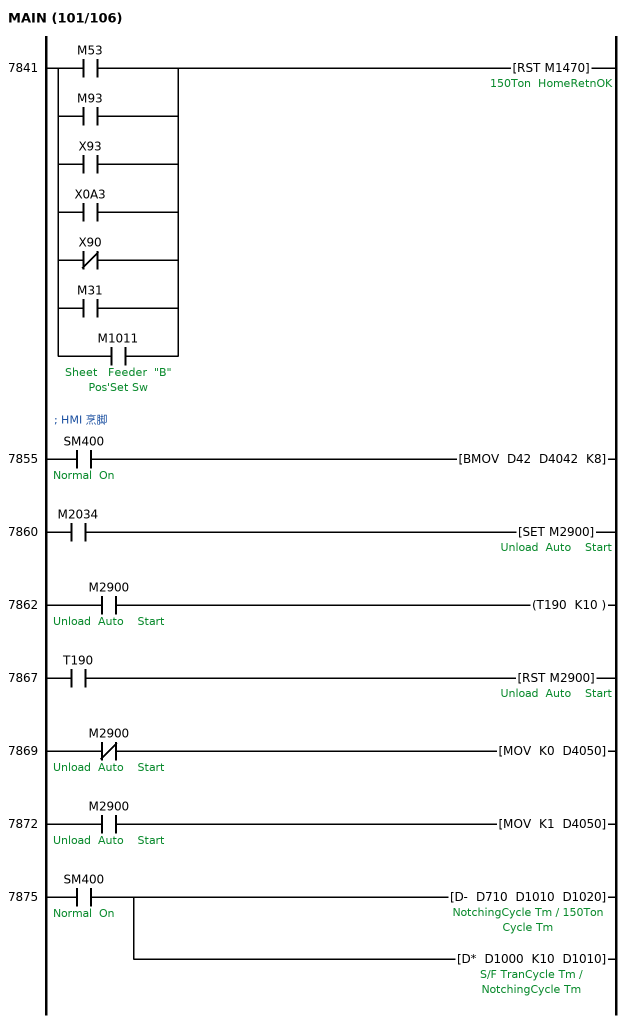
7841  LD      M53
      OR      M93
      OR      X93
      OR      X0A3
      ORI     X90
      OR      M31
      OR      M1011  ; Sheet   Feeder  "B" Pos'Set Sw
      RST     M1470  ; 150Ton  HomeRetnOK
; HMI 통신
7855  LD      SM400  ; Normal  On
      BMOV    D42 D4042 K8
7860  LD      M2034
      SET     M2900  ; Unload  Auto    Start
7862  LD      M2900  ; Unload  Auto    Start
      OUT     T190 K10
7867  LD      T190
      RST     M2900  ; Unload  Auto    Start
7869  LDI     M2900  ; Unload  Auto    Start
      MOV     K0 D4050
7872  LD      M2900  ; Unload  Auto    Start
      MOV     K1 D4050
7875  LD      SM400  ; Normal  On
      D-      D710 D1010 D1020  ; NotchingCycle Tm / 150Ton  Cycle Tm
      D*      D1000 K10 D1010  ; S/F TranCycle Tm
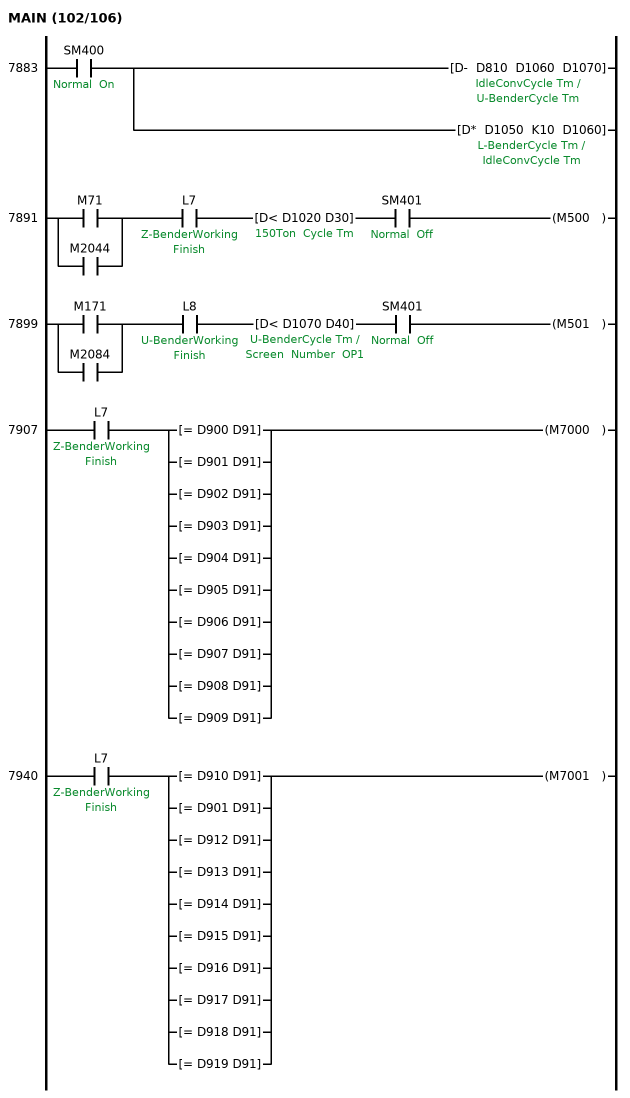
7883  LD      SM400  ; Normal  On
      D-      D810 D1060 D1070  ; IdleConvCycle Tm / U-BenderCycle Tm
      D*      D1050 K10 D1060  ; L-BenderCycle Tm
7891  LD      M71
      OR      M2044
      AND     L7  ; Z-BenderWorking Finish
      ANDD<   D1020 D30  ; 150Ton  Cycle Tm
      AND     SM401  ; Normal  Off
      OUT     M500
7899  LD      M171
      OR      M2084
      AND     L8  ; U-BenderWorking Finish
      ANDD<   D1070 D40  ; U-BenderCycle Tm / Screen  Number  OP1
      AND     SM401  ; Normal  Off
      OUT     M501
7907  LD      L7  ; Z-BenderWorking Finish
      LD=     D900 D91
      OR=     D901 D91
      OR=     D902 D91
      OR=     D903 D91
      OR=     D904 D91
      OR=     D905 D91
      OR=     D906 D91
      OR=     D907 D91
      OR=     D908 D91
      OR=     D909 D91
      ANB
      OUT     M7000
7940  LD      L7  ; Z-BenderWorking Finish
      LD=     D910 D91
      OR=     D901 D91
      OR=     D912 D91
      OR=     D913 D91
      OR=     D914 D91
      OR=     D915 D91
      OR=     D916 D91
      OR=     D917 D91
      OR=     D918 D91
      OR=     D919 D91
      ANB
      OUT     M7001
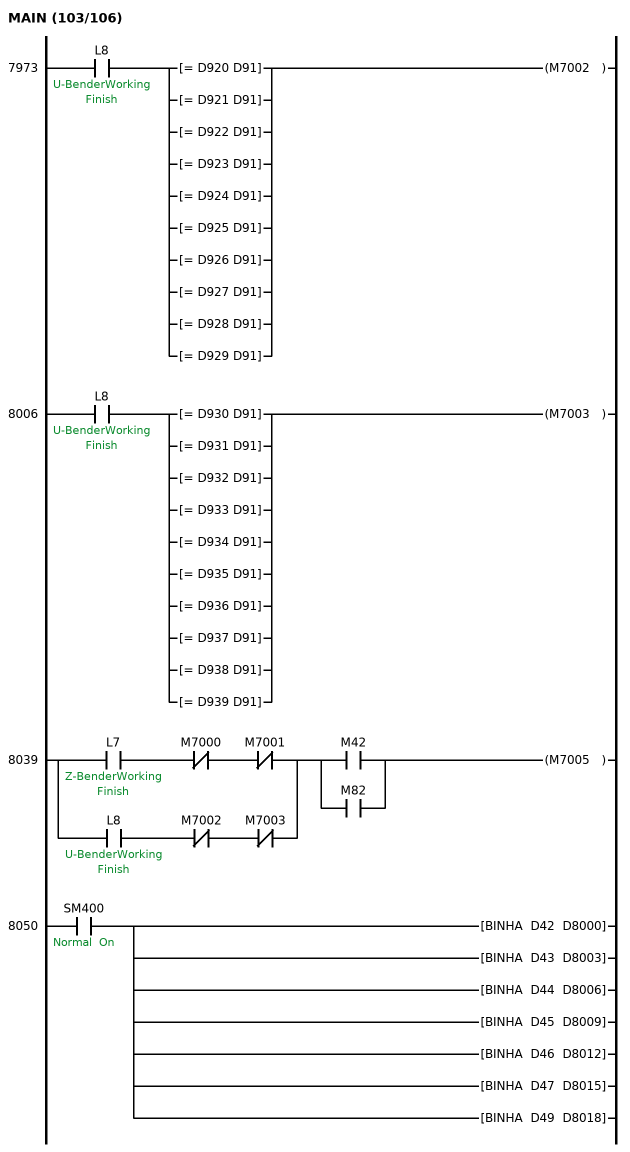
7973  LD      L8  ; U-BenderWorking Finish
      LD=     D920 D91
      OR=     D921 D91
      OR=     D922 D91
      OR=     D923 D91
      OR=     D924 D91
      OR=     D925 D91
      OR=     D926 D91
      OR=     D927 D91
      OR=     D928 D91
      OR=     D929 D91
      ANB
      OUT     M7002
8006  LD      L8  ; U-BenderWorking Finish
      LD=     D930 D91
      OR=     D931 D91
      OR=     D932 D91
      OR=     D933 D91
      OR=     D934 D91
      OR=     D935 D91
      OR=     D936 D91
      OR=     D937 D91
      OR=     D938 D91
      OR=     D939 D91
      ANB
      OUT     M7003
8039  LD      L7  ; Z-BenderWorking Finish
      ANI     M7000
      ANI     M7001
      LD      L8  ; U-BenderWorking Finish
      ANI     M7002
      ANI     M7003
      ORB
      LD      M42
      OR      M82
      ANB
      OUT     M7005
8050  LD      SM400  ; Normal  On
      BINHA   D42 D8000
      BINHA   D43 D8003
      BINHA   D44 D8006
      BINHA   D45 D8009
      BINHA   D46 D8012
      BINHA   D47 D8015
      BINHA   D49 D8018
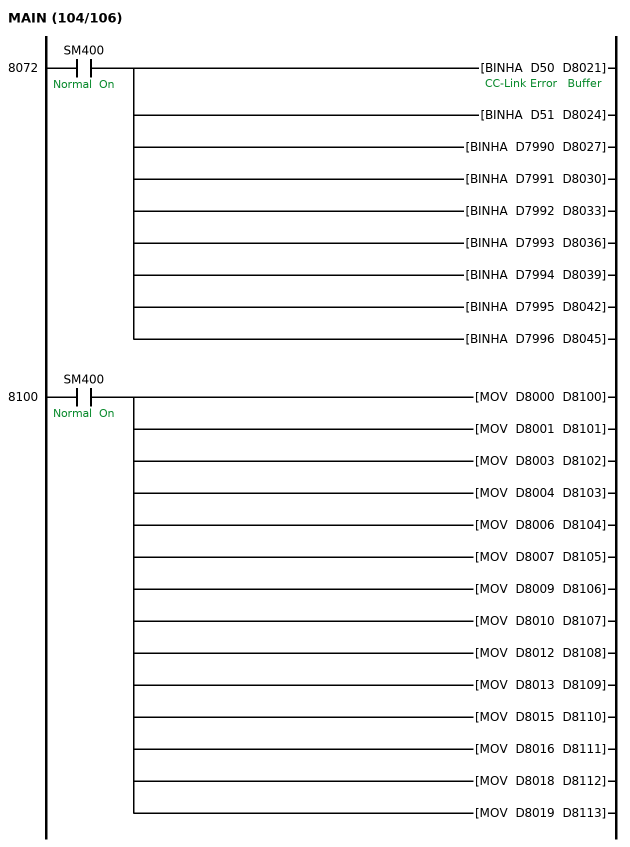
8072  LD      SM400  ; Normal  On
      BINHA   D50 D8021
      BINHA   D51 D8024
      BINHA   D7990 D8027
      BINHA   D7991 D8030
      BINHA   D7992 D8033
      BINHA   D7993 D8036
      BINHA   D7994 D8039
      BINHA   D7995 D8042
      BINHA   D7996 D8045
8100  LD      SM400  ; Normal  On
      MOV     D8000 D8100
      MOV     D8001 D8101
      MOV     D8003 D8102
      MOV     D8004 D8103
      MOV     D8006 D8104
      MOV     D8007 D8105
      MOV     D8009 D8106
      MOV     D8010 D8107
      MOV     D8012 D8108
      MOV     D8013 D8109
      MOV     D8015 D8110
      MOV     D8016 D8111
      MOV     D8018 D8112
      MOV     D8019 D8113
